TYPE ST_LoggerSettings :
STRUCT
	eLogLevelMinimum:		E_LogLevel:= E_LogLevel.Debug;
	eLogLevelMaximum:		E_LogLevel:= E_LogLevel.Critical;
END_STRUCT
END_TYPE

(* stored: Version 1.1.0.1
   DUT ST_LoggerSettings: Id {138d5e95-86ec-04dd-398b-aa4b90656350} *)
